{attribute 'pack_mode' := '1'}
TYPE ST_GetCellIndexDataIn :
STRUCT
	sCellID						: STRING(30);
END_STRUCT
END_TYPE

(* stored: Version 1.1.0.1, ProductVersion 3.1.4024.5
   DUT ST_GetCellIndexDataIn: Id {bbff5030-bc3b-4f39-8bb5-e4f0288f01fb} *)
